# EPICS substitutions: epics_iocs/GaussMeter/group5App/Db/magnet.substitutions
file "db/magnet.db" {
    pattern 	{ group, device }

    		{"group5", "GM"}
}
